Universal Robots URScript: hello.urscript

def test():
  textmsg("Hello world")
end
